FUNCTION_BLOCK Pocket (* Service Interface Function Block Type *)
  (* Standard: 61499-2; Description: Converts an AP224 machining feature into G code to be executed into FAGOR 8070 CNC controller *)
  (* Version 0.0, 2014-07-15, Esteban, ESID-UJI *)
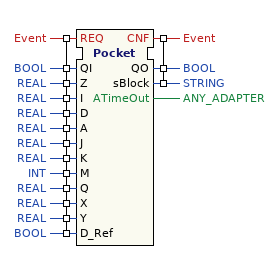
  EVENT_INPUT
    REQ WITH QI, Z, I, D, A, J, K, M, Q, X, Y, D_Ref; (* Service Request *)
  END_EVENT
  EVENT_OUTPUT
    CNF WITH QO, sBlock; (* Confirmation of Requested Service *)
  END_EVENT
  VAR_INPUT
    QI : BOOL; (* Event Input Qualifier *)
    Z : REAL; (* Reference plane *)
    I : REAL; (* pocket depth *)
    D : REAL; (* surface - reference plane distance *)
    A : REAL; (* angel with X-axis *)
    J : REAL; (* pocket half length *)
    K : REAL; (* pocket half width *)
    M : INT; (* Corner type *)
    Q : REAL; (* rounding radius *)
    X : REAL; (* X center position *)
    Y : REAL; (* Y center position *)
    D_Ref : BOOL := True; (* G90(F) or G91(T) *)
  END_VAR
  VAR_OUTPUT
    QO : BOOL; (* Event Output Qualifier *)
    sBlock : STRING; (* G code block *)
  END_VAR
  PLUGS
    ATimeOut : ANY_ADAPTER;
  END_PLUGS
  SERVICE APPLICATION/RESOURCE (* Service Interface Function Block Type *)
    SEQUENCE request_error
      APPLICATION.REQ+(SD) -> APPLICATION.CNF-(STATUS);
    END_SEQUENCE
    SEQUENCE request_inhibited
      APPLICATION.REQ-(SD) -> APPLICATION.CNF-(STATUS);
    END_SEQUENCE
    SEQUENCE request_confirm
      APPLICATION.REQ+(SD) -> APPLICATION.CNF+(RD);
    END_SEQUENCE
  END_SERVICE
END_FUNCTION_BLOCK
